// TIA Portal V17 export
// export: Created 2024-09-02T12:50:18.8272071Z, ExportSetting WithDefaults, DisplayName Totally Integrated Automation Portal, DisplayVersion V17, DisplayName TIA Portal Openness, DisplayVersion V17, DisplayName TIA Portal Version Control Interface, DisplayVersion V17, DisplayName STEP 7 Professional, DisplayVersion V17, DisplayName STEP 7 Safety, DisplayVersion V17, DisplayName WinCC Professional, DisplayVersion V17
DATA_BLOCK "DI_MachineOverview_Shift_Model_OP70"   // DB9
{ DB_Accessible_From_OPC_UA := 'FALSE' }
// stored: AutoNumber true, DBAccessibleFromOPCUA false, InstanceOfName FB_MachineOverview_Shift_Model, InstanceOfType FB
"FB_MachineOverview_Shift_Model"
   // VAR_INPUT
   //    FirstScan : Bool;
   //    PulseWorkpiece : Bool;
   // END_VAR
   // VAR_OUTPUT
   //    NumberOfPiecesActual : Int;
   //    UtilizationActual : Int;
   // END_VAR
   // VAR
   //    statRetVal_RD_LOC_T { ExternalAccessible := 'False'; ExternalVisible := 'False'; ExternalWritable := 'False'} : Int;
   //    statDateTimeLocalPLC { ExternalAccessible := 'False'; ExternalVisible := 'False'; ExternalWritable := 'False'} : DTL;
   //    statTimeOfDayPLC : Time_Of_Day;
   //    statWeekDayEurope : UInt;
   //    statDayInTheYear : UInt;
   //    statCalenderWeek : UInt;
   //    statSaveDay : USInt;
   //    statActShiftTimeRelativ : Real;
   //    statShift : Array[1..3] of Struct
   //       StartTime : Time_Of_Day;
   //       EndTime : Time_Of_Day;
   //       Pause : Time;
   //       Length : Time;
   //       Activ : Bool;
   //    END_STRUCT;
   // END_VAR
   // VAR RETAIN
   //    StatCurrentDayActiveShift : Byte;
   //    StatWeekDayActiveShift : USInt;
   //    StatCurrentShift : USInt;
   //    StatSaveShiftNumber : Byte;
   //    StatSavePulseWorkpiece : Bool;
   //    StatPulseWorkpiece : Bool;
   //    StatShiftChange : Bool;
   //    StatCWChange : Bool;
   //    Week : Array[0..2] of Struct
   //       CalenderWeek : Int;
   //       TargetShift1 : Int;
   //       TargetShift2 : Int;
   //       TargetShift3 : Int;
   //       TargetTotal : Int;
   //       NoOfPiecesTotal : Int;
   //       Weekday : Array[1..7] of Struct
   //          Day : Int;
   //          NoOfPieces : Int;
   //          Shift : Array[1..3] of Struct
   //             NoOfPieces : Int;
   //             "%" : Int;
   //          END_STRUCT;
   //       END_STRUCT;
   //    END_STRUCT;
   // END_VAR
   // VAR
   //    HMI_MachineUtilization : Struct
   //       "Week-" : Bool;
   //       "Week+" : Bool;
   //       "Pieces/Percent" : Bool;
   //       SelectedWeek : Int;
   //       WeekDay : Byte;
   //       Shift : Byte;
   //       WeekData : Struct
   //          CalenderWeek : Int;
   //          TargetShift1 : Int;
   //          TargetShift2 : Int;
   //          TargetShift3 : Int;
   //          TargetTotal : Int;
   //          NoOfPiecesTotal : Int;
   //          Weekday : Array[1..7] of Struct
   //             Day : Int;
   //             NoOfPieces : Int;
   //             Shift : Array[1..3] of Struct
   //                NoOfPieces : Int;
   //                "%" : Int;
   //             END_STRUCT;
   //          END_STRUCT;
   //       END_STRUCT;
   //    END_STRUCT;
   // END_VAR
   // VAR RETAIN
   //    HMI_ShiftModel : Struct
   //       CalenderWeek : Byte;
   //       WeekDay : Byte;
   //       DateTime : Date_And_Time;
   //       Shift : Array[1..3] of Struct
   //          StartTimeHour : USInt;
   //          StartTimeMinute : USInt;
   //          EndTimeHour : USInt;
   //          EndTimeMinute : USInt;
   //          PauseHour : USInt;
   //          PauseMinute : USInt;
   //          TargetShift : DInt;
   //       END_STRUCT;
   //       TargetCycleTime : Real;
   //       PartsPerCycle : Int;
   //       TargetOEE : Real;
   //       SetValues : Bool;
   //    END_STRUCT;
   // END_VAR
BEGIN
END_DATA_BLOCK
